// TIA Portal V20 export
ORGANIZATION_BLOCK "Startup"   // OB129, LAD, Startup
TITLE = "Complete Restart"
// stored: Namespace CITI_Logic, SetENOAutomatically false
   VAR_INPUT
      LostRetentive : Bool;   // True if retentive data are lost
      LostRTC : Bool;   // True if date and time are lost
   END_VAR
BEGIN
END_ORGANIZATION_BLOCK
